Universal Robots PolyScope program: Swan.urp

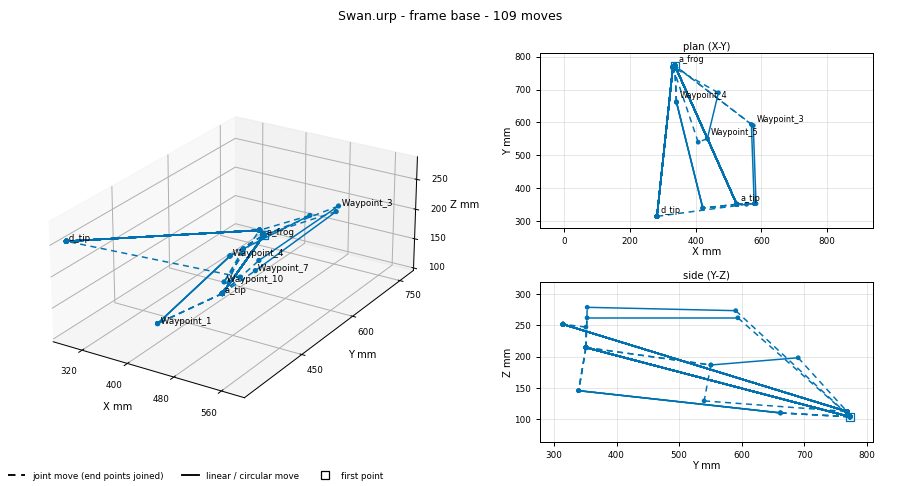
[picture p0: tool path of Swan.urp in frame base, 109 of 109 moves have a stored position in this frame; points joined in program order, loops and branches not executed]
Program Swan (installation=string_planes directory=/programs createdIn=5.17.3 lastSavedIn=5.17.3 robotSerialNumber=20245501435)
Calibrated DH parameters: a=[0.000154, -0.137004, -0.385524, -0.00002, 0.000092, 0]; d=[0.162441, 211.794786, -230.585024, 18.923638, 0.099786, 0.09951]; alpha=[1.569493, -0.001902, 0.003874, 1.570111, -1.570167, 0]; deltaTheta=[0, -1.242934, 1.056292, 0.186646, 0.000002, 0.000001]
InitVariablesNode
Robot Program (runOnlyOnce=true)
  SuppressedNode
    Wait Sleep waitTime=20
  Timer (action=Start) variable(name=beats)
  MoveL speed 150 mm/s, acceleration 600 mm/s^2 (useActiveTCP=true) feature=Base
    Waypoint a_frog: TCP in base x=336.638 y=773.336 z=103.937 mm, rx=-1.3698 ry=-2.3362 rz=1.327 rad; joints [-127.102, -6.181, 18.995, -50.118, -88.699, -156.884] deg; TCP offset x=28.21 y=-96.107 z=-99.69 mm, rx=0 ry=0 rz=0 rad
    Waypoint a_tip: TCP in base x=525.206 y=350.983 z=214.78 mm, rx=-1.3698 ry=-2.3362 rz=1.327 rad; joints [-161.028, -44.56, 81.191, -78.693, -115.03, -178.818] deg
      Until EXPRESSION (allowActions=false) ExpressionBranch=beats≥3
    Timer (action=Reset) variable=beats
  MoveJ speed 60 deg/s, acceleration 80 deg/s^2 (useActiveTCP=true) feature=Base
    Waypoint Waypoint_1: TCP in base x=421.786 y=339.391 z=145.77 mm, rx=-1.4848 ry=-2.1696 rz=1.0787 rad; joints [-159.235, -47.179, 101.918, -97.789, -99.401, -176.138] deg
  Timer (action=Reset) variable=beats
  MoveL speed 150 mm/s, acceleration 500 mm/s^2 (useActiveTCP=true) feature=Base
    Waypoint Waypoint_4: TCP in base x=341.564 y=662.071 z=110.192 mm, rx=-1.458 ry=-2.1893 rz=0.9879 rad; joints [-132.282, -25.96, 62.515, -82.619, -77.894, -159.669] deg
      Until EXPRESSION (allowActions=false) ExpressionBranch=beats≥3
  MoveJ speed 60 deg/s, acceleration 80 deg/s^2 (useActiveTCP=true) feature=Base
    Waypoint a_frog: TCP in base x=336.638 y=773.336 z=103.937 mm, rx=-1.3698 ry=-2.3362 rz=1.327 rad; joints [-127.102, -6.181, 18.995, -50.118, -88.699, -156.884] deg
  Timer (action=Reset) variable=beats
  MoveL speed 100 mm/s, acceleration 300 mm/s^2 (useActiveTCP=true) feature=Base
    Waypoint a_tip: motionParameters(blendRadius=0.03); TCP in base x=525.206 y=350.983 z=214.78 mm, rx=-1.3698 ry=-2.3362 rz=1.327 rad; joints [-161.028, -44.56, 81.191, -78.693, -115.03, -178.818] deg
      Until EXPRESSION (allowActions=false) ExpressionBranch=beats≥2.5
  Timer (action=Reset) variable=beats
  MoveL speed 400 mm/s, acceleration 1200 mm/s^2 (useActiveTCP=true) feature=Base
    Waypoint a_frog: TCP in base x=336.638 y=773.336 z=103.937 mm, rx=-1.3698 ry=-2.3362 rz=1.327 rad; joints [-127.102, -6.181, 18.995, -50.118, -88.699, -156.884] deg
      Until EXPRESSION (allowActions=false) ExpressionBranch=beats≥0.5
  Timer (action=Reset) variable=beats
  MoveL speed 100 mm/s, acceleration 600 mm/s^2 (useActiveTCP=true) feature=Base
    Waypoint a_tip: motionParameters(blendRadius=0.03); TCP in base x=525.206 y=350.983 z=214.78 mm, rx=-1.3698 ry=-2.3362 rz=1.327 rad; joints [-161.028, -44.56, 81.191, -78.693, -115.03, -178.818] deg
      Until EXPRESSION (allowActions=false) ExpressionBranch=beats≥2
  SuppressedNode
    Wait Sleep waitTime=21
  MoveJ speed 60 deg/s, acceleration 80 deg/s^2 (useActiveTCP=true) feature=Base
    Waypoint Waypoint_5: TCP in base x=435.657 y=550.869 z=186.821 mm, rx=-1.3927 ry=-2.3599 rz=1.285 rad; joints [-143.387, -35.735, 67.715, -72.278, -101.384, -166.853] deg
  MoveJ speed 60 deg/s, acceleration 80 deg/s^2 (useActiveTCP=true) feature=Base
    Waypoint Waypoint_10: TCP in base x=407.775 y=540.024 z=129.396 mm, rx=-1.4447 ry=-1.9576 rz=1.0842 rad; joints [-142.798, -34.554, 77.92, -79.333, -77.889, -165.949] deg
  SuppressedNode
    MoveL speed 400 mm/s, acceleration 1200 mm/s^2 (useActiveTCP=true) feature=Base
      Waypoint Waypoint_6: TCP in base x=469.305 y=690.432 z=198.38 mm, rx=-1.3698 ry=-2.3362 rz=1.327 rad; joints [-137.273, -11.027, 15.189, -41.782, -96.797, -163.098] deg
  MoveJ speed 60 deg/s, acceleration 80 deg/s^2 (useActiveTCP=true) feature=Base
    Waypoint d_frog: TCP in base x=330.848 y=768.457 z=112.523 mm, rx=-1.919 ry=-1.7189 rz=1.2902 rad; joints [-128.404, -20.72, 47.39, -64.46, -68.674, -132.513] deg
  Timer (action=Reset) variable=beats
  MoveL speed 200 mm/s, acceleration 600 mm/s^2 (useActiveTCP=true) feature=Base
    Waypoint d_tip: TCP in base x=282.292 y=314.303 z=251.965 mm, rx=-1.8973 ry=-1.7705 rz=1.2029 rad; joints [-160.183, -75.446, 125.19, -87.671, -93.352, -154.437] deg
      Until EXPRESSION (allowActions=false) ExpressionBranch=beats≥2
  Timer (action=Reset) variable=beats
  Timer (action=Start) variable=beats
  MoveL speed 150 mm/s, acceleration 600 mm/s^2 (useActiveTCP=true) feature=Base
    Waypoint d_frog: TCP in base x=330.848 y=768.457 z=112.523 mm, rx=-1.919 ry=-1.7189 rz=1.2902 rad; joints [-128.404, -20.72, 47.39, -64.46, -68.674, -132.513] deg
      Until EXPRESSION (allowActions=false) ExpressionBranch=beats≥0.5
  Timer (action=Reset) variable=beats
  MoveL speed 150 mm/s, acceleration 600 mm/s^2 (useActiveTCP=true) feature=Base
    Waypoint d_tip: TCP in base x=282.292 y=314.303 z=251.965 mm, rx=-1.8973 ry=-1.7705 rz=1.2029 rad; joints [-160.183, -75.446, 125.19, -87.671, -93.352, -154.437] deg
      Until EXPRESSION (allowActions=false) ExpressionBranch=beats≥0.5
  Timer (action=Reset) variable=beats
  MoveL speed 150 mm/s, acceleration 600 mm/s^2 (useActiveTCP=true) feature=Base
    Waypoint d_frog: TCP in base x=330.848 y=768.457 z=112.523 mm, rx=-1.919 ry=-1.7189 rz=1.2902 rad; joints [-128.404, -20.72, 47.39, -64.46, -68.674, -132.513] deg
      Until EXPRESSION (allowActions=false) ExpressionBranch=beats≥0.5
  Timer (action=Reset) variable=beats
  MoveL speed 150 mm/s, acceleration 600 mm/s^2 (useActiveTCP=true) feature=Base
    Waypoint d_tip: TCP in base x=282.292 y=314.303 z=251.965 mm, rx=-1.8973 ry=-1.7705 rz=1.2029 rad; joints [-160.183, -75.446, 125.19, -87.671, -93.352, -154.437] deg
      Until EXPRESSION (allowActions=false) ExpressionBranch=beats≥0.5
  Timer (action=Reset) variable=beats
  MoveL speed 150 mm/s, acceleration 600 mm/s^2 (useActiveTCP=true) feature=Base
    Waypoint d_frog: TCP in base x=330.848 y=768.457 z=112.523 mm, rx=-1.919 ry=-1.7189 rz=1.2902 rad; joints [-128.404, -20.72, 47.39, -64.46, -68.674, -132.513] deg
      Until EXPRESSION (allowActions=false) ExpressionBranch=beats≥0.5
  Timer (action=Reset) variable=beats
  MoveL speed 150 mm/s, acceleration 600 mm/s^2 (useActiveTCP=true) feature=Base
    Waypoint d_tip: TCP in base x=282.292 y=314.303 z=251.965 mm, rx=-1.8973 ry=-1.7705 rz=1.2029 rad; joints [-160.183, -75.446, 125.19, -87.671, -93.352, -154.437] deg
      Until EXPRESSION (allowActions=false) ExpressionBranch=beats≥0.5
  Timer (action=Reset) variable=beats
  MoveL speed 150 mm/s, acceleration 600 mm/s^2 (useActiveTCP=true) feature=Base
    Waypoint d_frog: TCP in base x=330.848 y=768.457 z=112.523 mm, rx=-1.919 ry=-1.7189 rz=1.2902 rad; joints [-128.404, -20.72, 47.39, -64.46, -68.674, -132.513] deg
      Until EXPRESSION (allowActions=false) ExpressionBranch=beats≥0.5
  Timer (action=Reset) variable=beats
  MoveL speed 150 mm/s, acceleration 600 mm/s^2 (useActiveTCP=true) feature=Base
    Waypoint d_tip: TCP in base x=282.292 y=314.303 z=251.965 mm, rx=-1.8973 ry=-1.7705 rz=1.2029 rad; joints [-160.183, -75.446, 125.19, -87.671, -93.352, -154.437] deg
      Until EXPRESSION (allowActions=false) ExpressionBranch=beats≥0.5
  Timer (action=Reset) variable=beats
  MoveL speed 150 mm/s, acceleration 600 mm/s^2 (useActiveTCP=true) feature=Base
    Waypoint d_frog: TCP in base x=330.848 y=768.457 z=112.523 mm, rx=-1.919 ry=-1.7189 rz=1.2902 rad; joints [-128.404, -20.72, 47.39, -64.46, -68.674, -132.513] deg
      Until EXPRESSION (allowActions=false) ExpressionBranch=beats≥3.5
  MoveJ speed 60 deg/s, acceleration 80 deg/s^2 (useActiveTCP=true) feature=Base
    Waypoint a_frog: TCP in base x=336.638 y=773.336 z=103.937 mm, rx=-1.3698 ry=-2.3362 rz=1.327 rad; joints [-127.102, -6.181, 18.995, -50.118, -88.699, -156.884] deg
  Wait Sleep waitTime=1
  Timer (action=Reset) variable=beats
  MoveL speed 150 mm/s, acceleration 600 mm/s^2 (useActiveTCP=true) feature=Base
    Waypoint a_frog: TCP in base x=336.638 y=773.336 z=103.937 mm, rx=-1.3698 ry=-2.3362 rz=1.327 rad; joints [-127.102, -6.181, 18.995, -50.118, -88.699, -156.884] deg
    Waypoint a_tip: TCP in base x=525.206 y=350.983 z=214.78 mm, rx=-1.3698 ry=-2.3362 rz=1.327 rad; joints [-161.028, -44.56, 81.191, -78.693, -115.03, -178.818] deg
      Until EXPRESSION (allowActions=false) ExpressionBranch=beats≥3
    Timer (action=Reset) variable=beats
  MoveJ speed 60 deg/s, acceleration 80 deg/s^2 (useActiveTCP=true) feature=Base
    Waypoint Waypoint_1: TCP in base x=421.786 y=339.391 z=145.77 mm, rx=-1.4848 ry=-2.1696 rz=1.0787 rad; joints [-159.235, -47.179, 101.918, -97.789, -99.401, -176.138] deg
  Timer (action=Reset) variable=beats
  MoveL speed 150 mm/s, acceleration 500 mm/s^2 (useActiveTCP=true) feature=Base
    Waypoint Waypoint_4: TCP in base x=341.564 y=662.071 z=110.192 mm, rx=-1.458 ry=-2.1893 rz=0.9879 rad; joints [-132.282, -25.96, 62.515, -82.619, -77.894, -159.669] deg
      Until EXPRESSION (allowActions=false) ExpressionBranch=beats≥3
  MoveJ speed 60 deg/s, acceleration 80 deg/s^2 (useActiveTCP=true) feature=Base
    Waypoint a_frog: TCP in base x=336.638 y=773.336 z=103.937 mm, rx=-1.3698 ry=-2.3362 rz=1.327 rad; joints [-127.102, -6.181, 18.995, -50.118, -88.699, -156.884] deg
  MoveL speed 100 mm/s, acceleration 300 mm/s^2 (useActiveTCP=true) feature=Base
    Waypoint a_tip: motionParameters(blendRadius=0.03); TCP in base x=525.206 y=350.983 z=214.78 mm, rx=-1.3698 ry=-2.3362 rz=1.327 rad; joints [-161.028, -44.56, 81.191, -78.693, -115.03, -178.818] deg
      Until EXPRESSION (allowActions=false) ExpressionBranch=beats≥2.5
  Timer (action=Reset) variable=beats
  MoveL speed 250 mm/s, acceleration 1200 mm/s^2 (useActiveTCP=true) feature=Base
    Waypoint a_frog: TCP in base x=336.638 y=773.336 z=103.937 mm, rx=-1.3698 ry=-2.3362 rz=1.327 rad; joints [-127.102, -6.181, 18.995, -50.118, -88.699, -156.884] deg
      Until EXPRESSION (allowActions=false) ExpressionBranch=beats≥0.5
  Timer (action=Reset) variable=beats
  MoveL speed 100 mm/s, acceleration 600 mm/s^2 (useActiveTCP=true) feature=Base
    Waypoint a_tip: motionParameters(blendRadius=0.03); TCP in base x=525.206 y=350.983 z=214.78 mm, rx=-1.3698 ry=-2.3362 rz=1.327 rad; joints [-161.028, -44.56, 81.191, -78.693, -115.03, -178.818] deg
      Until EXPRESSION (allowActions=false) ExpressionBranch=beats≥3
  MoveJ speed 60 deg/s, acceleration 80 deg/s^2 (useActiveTCP=true) feature=Base
    Waypoint Waypoint_9: TCP in base x=554.848 y=350.983 z=247.422 mm, rx=-1.3698 ry=-2.3362 rz=1.327 rad; joints [-161.804, -44.051, 74.534, -72.804, -115.615, -179.417] deg
  MoveJ speed 60 deg/s, acceleration 80 deg/s^2 (useActiveTCP=true) feature=Base
    Waypoint d_tip: TCP in base x=282.292 y=314.303 z=251.965 mm, rx=-1.8973 ry=-1.7705 rz=1.2029 rad; joints [-160.183, -75.446, 125.19, -87.671, -93.352, -154.437] deg
  Timer (action=Reset) variable=beats
  Timer (action=Start) variable=beats
  MoveL speed 150 mm/s, acceleration 60 mm/s^2 (useActiveTCP=true) feature=Base
    Waypoint d_frog: TCP in base x=330.848 y=768.457 z=112.523 mm, rx=-1.919 ry=-1.7189 rz=1.2902 rad; joints [-128.404, -20.72, 47.39, -64.46, -68.674, -132.513] deg
      Until EXPRESSION (allowActions=false) ExpressionBranch=beats≥1.5
  Timer (action=Reset) variable=beats
  Timer (action=Start) variable=beats
  MoveL speed 150 mm/s, acceleration 600 mm/s^2 (useActiveTCP=true) feature=Base
    Waypoint d_tip: TCP in base x=282.292 y=314.303 z=251.965 mm, rx=-1.8973 ry=-1.7705 rz=1.2029 rad; joints [-160.183, -75.446, 125.19, -87.671, -93.352, -154.437] deg
      Until EXPRESSION (allowActions=false) ExpressionBranch=beats≥0.5
  Timer (action=Reset) variable=beats
  MoveL speed 150 mm/s, acceleration 600 mm/s^2 (useActiveTCP=true) feature=Base
    Waypoint d_frog: TCP in base x=330.848 y=768.457 z=112.523 mm, rx=-1.919 ry=-1.7189 rz=1.2902 rad; joints [-128.404, -20.72, 47.39, -64.46, -68.674, -132.513] deg
      Until EXPRESSION (allowActions=false) ExpressionBranch=beats≥0.5
  Timer (action=Reset) variable=beats
  MoveL speed 150 mm/s, acceleration 600 mm/s^2 (useActiveTCP=true) feature=Base
    Waypoint d_tip: TCP in base x=282.292 y=314.303 z=251.965 mm, rx=-1.8973 ry=-1.7705 rz=1.2029 rad; joints [-160.183, -75.446, 125.19, -87.671, -93.352, -154.437] deg
      Until EXPRESSION (allowActions=false) ExpressionBranch=beats≥0.5
  Timer (action=Reset) variable=beats
  MoveL speed 150 mm/s, acceleration 600 mm/s^2 (useActiveTCP=true) feature=Base
    Waypoint d_frog: TCP in base x=330.848 y=768.457 z=112.523 mm, rx=-1.919 ry=-1.7189 rz=1.2902 rad; joints [-128.404, -20.72, 47.39, -64.46, -68.674, -132.513] deg
      Until EXPRESSION (allowActions=false) ExpressionBranch=beats≥0.5
  Timer (action=Reset) variable=beats
  MoveL speed 150 mm/s, acceleration 600 mm/s^2 (useActiveTCP=true) feature=Base
    Waypoint d_tip: TCP in base x=282.292 y=314.303 z=251.965 mm, rx=-1.8973 ry=-1.7705 rz=1.2029 rad; joints [-160.183, -75.446, 125.19, -87.671, -93.352, -154.437] deg
      Until EXPRESSION (allowActions=false) ExpressionBranch=beats≥0.5
  Timer (action=Reset) variable=beats
  MoveL speed 150 mm/s, acceleration 600 mm/s^2 (useActiveTCP=true) feature=Base
    Waypoint d_frog: TCP in base x=330.848 y=768.457 z=112.523 mm, rx=-1.919 ry=-1.7189 rz=1.2902 rad; joints [-128.404, -20.72, 47.39, -64.46, -68.674, -132.513] deg
      Until EXPRESSION (allowActions=false) ExpressionBranch=beats≥0.5
  Timer (action=Reset) variable=beats
  MoveL speed 150 mm/s, acceleration 600 mm/s^2 (useActiveTCP=true) feature=Base
    Waypoint d_tip: TCP in base x=282.292 y=314.303 z=251.965 mm, rx=-1.8973 ry=-1.7705 rz=1.2029 rad; joints [-160.183, -75.446, 125.19, -87.671, -93.352, -154.437] deg
      Until EXPRESSION (allowActions=false) ExpressionBranch=beats≥0.5
  Timer (action=Reset) variable=beats
  MoveL speed 150 mm/s, acceleration 600 mm/s^2 (useActiveTCP=true) feature=Base
    Waypoint d_frog: TCP in base x=330.848 y=768.457 z=112.523 mm, rx=-1.919 ry=-1.7189 rz=1.2902 rad; joints [-128.404, -20.72, 47.39, -64.46, -68.674, -132.513] deg
      Until EXPRESSION (allowActions=false) ExpressionBranch=beats≥0.5
  Timer (action=Reset) variable=beats
  MoveL speed 100 mm/s, acceleration 500 mm/s^2 (useActiveTCP=true) feature=Base
    Waypoint d_frog: TCP in base x=330.848 y=768.457 z=112.523 mm, rx=-1.919 ry=-1.7189 rz=1.2902 rad; joints [-128.404, -20.72, 47.39, -64.46, -68.674, -132.513] deg
      Until EXPRESSION (allowActions=false) ExpressionBranch=beats≥3.5
  MoveJ speed 60 deg/s, acceleration 80 deg/s^2 (useActiveTCP=true) feature=Base
    Waypoint a_frog: TCP in base x=336.638 y=773.336 z=103.937 mm, rx=-1.3698 ry=-2.3362 rz=1.327 rad; joints [-127.102, -6.181, 18.995, -50.118, -88.699, -156.884] deg
  Wait Sleep waitTime=1
  Timer (action=Reset) variable=beats
  MoveL speed 150 mm/s, acceleration 600 mm/s^2 (useActiveTCP=true) feature=Base
    Waypoint a_frog: TCP in base x=336.638 y=773.336 z=103.937 mm, rx=-1.3698 ry=-2.3362 rz=1.327 rad; joints [-127.102, -6.181, 18.995, -50.118, -88.699, -156.884] deg
    Waypoint a_tip: TCP in base x=525.206 y=350.983 z=214.78 mm, rx=-1.3698 ry=-2.3362 rz=1.327 rad; joints [-161.028, -44.56, 81.191, -78.693, -115.03, -178.818] deg
      Until EXPRESSION (allowActions=false) ExpressionBranch=beats≥3
    Timer (action=Reset) variable=beats
  MoveL speed 100 mm/s, acceleration 600 mm/s^2 (useActiveTCP=true) feature=Base
    Waypoint a_frog: TCP in base x=336.638 y=773.336 z=103.937 mm, rx=-1.3698 ry=-2.3362 rz=1.327 rad; joints [-127.102, -6.181, 18.995, -50.118, -88.699, -156.884] deg
      Until EXPRESSION (allowActions=false) ExpressionBranch=beats≥3
  Timer (action=Reset) variable=beats
  MoveL speed 100 mm/s, acceleration 600 mm/s^2 (useActiveTCP=true) feature=Base
    Waypoint a_tip: TCP in base x=525.206 y=350.983 z=214.78 mm, rx=-1.3698 ry=-2.3362 rz=1.327 rad; joints [-161.028, -44.56, 81.191, -78.693, -115.03, -178.818] deg
      Until EXPRESSION (allowActions=false) ExpressionBranch=beats≥2.5
  Timer (action=Reset) variable=beats
  MoveL speed 300 mm/s, acceleration 1200 mm/s^2 (useActiveTCP=true) feature=Base
    Waypoint a_frog: TCP in base x=336.638 y=773.336 z=103.937 mm, rx=-1.3698 ry=-2.3362 rz=1.327 rad; joints [-127.102, -6.181, 18.995, -50.118, -88.699, -156.884] deg
      Until EXPRESSION (allowActions=false) ExpressionBranch=beats≥0.5
  MoveL speed 150 mm/s, acceleration 600 mm/s^2 (useActiveTCP=true) feature=Base
    Waypoint a_tip: TCP in base x=525.206 y=350.983 z=214.78 mm, rx=-1.3698 ry=-2.3362 rz=1.327 rad; joints [-161.028, -44.56, 81.191, -78.693, -115.03, -178.818] deg
      Until EXPRESSION (allowActions=false) ExpressionBranch=beats≥2
  MoveJ speed 60 deg/s, acceleration 80 deg/s^2 (useActiveTCP=true) feature=Base
    Waypoint Waypoint_2: TCP in base x=583.831 y=353.076 z=279.049 mm, rx=-1.3698 ry=-2.3362 rz=1.327 rad; joints [-162.353, -42.73, 66.875, -66.655, -116.033, -179.849] deg
  MoveL speed 400 mm/s, acceleration 1200 mm/s^2 (useActiveTCP=true) feature=Base
    Waypoint Waypoint_3: TCP in base x=575.353 y=590.579 z=273.677 mm, rx=-1.3698 ry=-2.3362 rz=1.327 rad; joints [-146.762, -11.123, 4.55, -32.162, -104.295, -169.078] deg
  MoveJ speed 60 deg/s, acceleration 80 deg/s^2 (useActiveTCP=true) feature=Base
    Waypoint a_frog: TCP in base x=336.638 y=773.336 z=103.937 mm, rx=-1.3698 ry=-2.3362 rz=1.327 rad; joints [-127.102, -6.181, 18.995, -50.118, -88.699, -156.884] deg
  MoveL speed 200 mm/s, acceleration 600 mm/s^2 (useActiveTCP=true) feature=Base
    Waypoint a_tip: TCP in base x=525.206 y=350.983 z=214.78 mm, rx=-1.3698 ry=-2.3362 rz=1.327 rad; joints [-161.028, -44.56, 81.191, -78.693, -115.03, -178.818] deg
      Until EXPRESSION (allowActions=false) ExpressionBranch=beats≥1
  Timer (action=Reset) variable=beats
  MoveL speed 200 mm/s, acceleration 600 mm/s^2 (useActiveTCP=true) feature=Base
    Waypoint a_frog: TCP in base x=336.638 y=773.336 z=103.937 mm, rx=-1.3698 ry=-2.3362 rz=1.327 rad; joints [-127.102, -6.181, 18.995, -50.118, -88.699, -156.884] deg
      Until EXPRESSION (allowActions=false) ExpressionBranch=beats≥1
  Timer (action=Reset) variable=beats
  MoveL speed 200 mm/s, acceleration 600 mm/s^2 (useActiveTCP=true) feature=Base
    Waypoint a_tip: TCP in base x=525.206 y=350.983 z=214.78 mm, rx=-1.3698 ry=-2.3362 rz=1.327 rad; joints [-161.028, -44.56, 81.191, -78.693, -115.03, -178.818] deg
      Until EXPRESSION (allowActions=false) ExpressionBranch=beats≥1
  Timer (action=Reset) variable=beats
  MoveL speed 200 mm/s, acceleration 600 mm/s^2 (useActiveTCP=true) feature=Base
    Waypoint a_frog: TCP in base x=336.638 y=773.336 z=103.937 mm, rx=-1.3698 ry=-2.3362 rz=1.327 rad; joints [-127.102, -6.181, 18.995, -50.118, -88.699, -156.884] deg
      Until EXPRESSION (allowActions=false) ExpressionBranch=beats≥1
  Timer (action=Reset) variable=beats
  MoveL speed 200 mm/s, acceleration 600 mm/s^2 (useActiveTCP=true) feature=Base
    Waypoint a_tip: TCP in base x=525.206 y=350.983 z=214.78 mm, rx=-1.3698 ry=-2.3362 rz=1.327 rad; joints [-161.028, -44.56, 81.191, -78.693, -115.03, -178.818] deg
      Until EXPRESSION (allowActions=false) ExpressionBranch=beats≥1
  Timer (action=Reset) variable=beats
  MoveL speed 250 mm/s, acceleration 600 mm/s^2 (useActiveTCP=true) feature=Base
    Waypoint a_frog: TCP in base x=336.638 y=773.336 z=103.937 mm, rx=-1.3698 ry=-2.3362 rz=1.327 rad; joints [-127.102, -6.181, 18.995, -50.118, -88.699, -156.884] deg
      Until EXPRESSION (allowActions=false) ExpressionBranch=beats≥1
  Timer (action=Reset) variable=beats
  MoveL speed 100 mm/s, acceleration 600 mm/s^2 (useActiveTCP=true) feature=Base
    Waypoint a_tip: TCP in base x=525.206 y=350.983 z=214.78 mm, rx=-1.3698 ry=-2.3362 rz=1.327 rad; joints [-161.028, -44.56, 81.191, -78.693, -115.03, -178.818] deg
      Until EXPRESSION (allowActions=false) ExpressionBranch=beats≥2.5
  Timer (action=Reset) variable=beats
  MoveL speed 250 mm/s, acceleration 1200 mm/s^2 (useActiveTCP=true) feature=Base
    Waypoint a_frog: TCP in base x=336.638 y=773.336 z=103.937 mm, rx=-1.3698 ry=-2.3362 rz=1.327 rad; joints [-127.102, -6.181, 18.995, -50.118, -88.699, -156.884] deg
      Until EXPRESSION (allowActions=false) ExpressionBranch=beats≥0.5
  Timer (action=Reset) variable=beats
  MoveL speed 150 mm/s, acceleration 600 mm/s^2 (useActiveTCP=true) feature=Base
    Waypoint a_tip: TCP in base x=525.206 y=350.983 z=214.78 mm, rx=-1.3698 ry=-2.3362 rz=1.327 rad; joints [-161.028, -44.56, 81.191, -78.693, -115.03, -178.818] deg
      Until EXPRESSION (allowActions=false) ExpressionBranch=beats≥2
  Timer (action=Reset) variable=beats
  MoveJ speed 60 deg/s, acceleration 80 deg/s^2 (useActiveTCP=true) feature=Base
    Waypoint Waypoint_7: TCP in base x=578.283 y=352.878 z=262.264 mm, rx=-1.3698 ry=-2.3362 rz=1.327 rad; joints [-162.237, -42.346, 68.857, -68.978, -115.943, -179.753] deg
  MoveL speed 400 mm/s, acceleration 1200 mm/s^2 (useActiveTCP=true) feature=Base
    Waypoint Waypoint_8: TCP in base x=569.678 y=593.931 z=262.264 mm, rx=-1.3698 ry=-2.3362 rz=1.327 rad; joints [-146.374, -13.725, 11.576, -36.522, -103.973, -168.824] deg
  MoveJ speed 60 deg/s, acceleration 80 deg/s^2 (useActiveTCP=true) feature=Base
    Waypoint a_frog: TCP in base x=336.638 y=773.336 z=103.937 mm, rx=-1.3698 ry=-2.3362 rz=1.327 rad; joints [-127.102, -6.181, 18.995, -50.118, -88.699, -156.884] deg
  Timer (action=Reset) variable=beats
  MoveL speed 200 mm/s, acceleration 600 mm/s^2 (useActiveTCP=true) feature=Base
    Waypoint a_tip: TCP in base x=525.206 y=350.983 z=214.78 mm, rx=-1.3698 ry=-2.3362 rz=1.327 rad; joints [-161.028, -44.56, 81.191, -78.693, -115.03, -178.818] deg
      Until EXPRESSION (allowActions=false) ExpressionBranch=beats≥1
  Timer (action=Reset) variable=beats
  MoveL speed 200 mm/s, acceleration 600 mm/s^2 (useActiveTCP=true) feature=Base
    Waypoint a_frog: TCP in base x=336.638 y=773.336 z=103.937 mm, rx=-1.3698 ry=-2.3362 rz=1.327 rad; joints [-127.102, -6.181, 18.995, -50.118, -88.699, -156.884] deg
      Until EXPRESSION (allowActions=false) ExpressionBranch=beats≥1
  Timer (action=Reset) variable=beats
  MoveL speed 200 mm/s, acceleration 600 mm/s^2 (useActiveTCP=true) feature=Base
    Waypoint a_tip: TCP in base x=525.206 y=350.983 z=214.78 mm, rx=-1.3698 ry=-2.3362 rz=1.327 rad; joints [-161.028, -44.56, 81.191, -78.693, -115.03, -178.818] deg
      Until EXPRESSION (allowActions=false) ExpressionBranch=beats≥1
  Timer (action=Reset) variable=beats
  MoveL speed 100 mm/s, acceleration 600 mm/s^2 (useActiveTCP=true) feature=Base
    Waypoint a_frog: TCP in base x=336.638 y=773.336 z=103.937 mm, rx=-1.3698 ry=-2.3362 rz=1.327 rad; joints [-127.102, -6.181, 18.995, -50.118, -88.699, -156.884] deg
      Until EXPRESSION (allowActions=false) ExpressionBranch=beats≥2
  Timer (action=Reset) variable=beats
  MoveL speed 250 mm/s, acceleration 1200 mm/s^2 (useActiveTCP=true) feature=Base
    Waypoint a_tip: TCP in base x=525.206 y=350.983 z=214.78 mm, rx=-1.3698 ry=-2.3362 rz=1.327 rad; joints [-161.028, -44.56, 81.191, -78.693, -115.03, -178.818] deg
      Until EXPRESSION (allowActions=false) ExpressionBranch=beats≥0.5
  Timer (action=Reset) variable=beats
  MoveL speed 250 mm/s, acceleration 1200 mm/s^2 (useActiveTCP=true) feature=Base
    Waypoint a_frog: TCP in base x=336.638 y=773.336 z=103.937 mm, rx=-1.3698 ry=-2.3362 rz=1.327 rad; joints [-127.102, -6.181, 18.995, -50.118, -88.699, -156.884] deg
      Until EXPRESSION (allowActions=false) ExpressionBranch=beats≥0.5
  Timer (action=Reset) variable=beats
  MoveL speed 150 mm/s, acceleration 600 mm/s^2 (useActiveTCP=true) feature=Base
    Waypoint a_tip: TCP in base x=525.206 y=350.983 z=214.78 mm, rx=-1.3698 ry=-2.3362 rz=1.327 rad; joints [-161.028, -44.56, 81.191, -78.693, -115.03, -178.818] deg
      Until EXPRESSION (allowActions=false) ExpressionBranch=beats≥3
  Timer (action=Reset) variable=beats
  MoveL speed 150 mm/s, acceleration 600 mm/s^2 (useActiveTCP=true) feature=Base
    Waypoint a_frog: TCP in base x=336.638 y=773.336 z=103.937 mm, rx=-1.3698 ry=-2.3362 rz=1.327 rad; joints [-127.102, -6.181, 18.995, -50.118, -88.699, -156.884] deg
      Until EXPRESSION (allowActions=false) ExpressionBranch=beats≥3
  Timer (action=Reset) variable=beats
  MoveL speed 150 mm/s, acceleration 600 mm/s^2 (useActiveTCP=true) feature=Base
    Waypoint a_tip: TCP in base x=525.206 y=350.983 z=214.78 mm, rx=-1.3698 ry=-2.3362 rz=1.327 rad; joints [-161.028, -44.56, 81.191, -78.693, -115.03, -178.818] deg
      Until EXPRESSION (allowActions=false) ExpressionBranch=beats≥3
  Timer (action=Reset) variable=beats
  MoveL speed 150 mm/s, acceleration 600 mm/s^2 (useActiveTCP=true) feature=Base
    Waypoint a_frog: TCP in base x=336.638 y=773.336 z=103.937 mm, rx=-1.3698 ry=-2.3362 rz=1.327 rad; joints [-127.102, -6.181, 18.995, -50.118, -88.699, -156.884] deg
      Until EXPRESSION (allowActions=false) ExpressionBranch=beats≥2
  Timer (action=Reset) variable=beats
  MoveL speed 250 mm/s, acceleration 1200 mm/s^2 (useActiveTCP=true) feature=Base
    Waypoint a_tip: TCP in base x=525.206 y=350.983 z=214.78 mm, rx=-1.3698 ry=-2.3362 rz=1.327 rad; joints [-161.028, -44.56, 81.191, -78.693, -115.03, -178.818] deg
      Until EXPRESSION (allowActions=false) ExpressionBranch=beats≥0.5
  Timer (action=Reset) variable=beats
  MoveL speed 250 mm/s, acceleration 1200 mm/s^2 (useActiveTCP=true) feature=Base
    Waypoint a_frog: TCP in base x=336.638 y=773.336 z=103.937 mm, rx=-1.3698 ry=-2.3362 rz=1.327 rad; joints [-127.102, -6.181, 18.995, -50.118, -88.699, -156.884] deg
      Until EXPRESSION (allowActions=false) ExpressionBranch=beats≥0.5
  Timer (action=Reset) variable=beats
  MoveL speed 150 mm/s, acceleration 600 mm/s^2 (useActiveTCP=true) feature=Base
    Waypoint a_tip: TCP in base x=525.206 y=350.983 z=214.78 mm, rx=-1.3698 ry=-2.3362 rz=1.327 rad; joints [-161.028, -44.56, 81.191, -78.693, -115.03, -178.818] deg
      Until EXPRESSION (allowActions=false) ExpressionBranch=beats≥3
  Timer (action=Reset) variable=beats
  MoveL speed 150 mm/s, acceleration 600 mm/s^2 (useActiveTCP=true) feature=Base
    Waypoint a_frog: TCP in base x=336.638 y=773.336 z=103.937 mm, rx=-1.3698 ry=-2.3362 rz=1.327 rad; joints [-127.102, -6.181, 18.995, -50.118, -88.699, -156.884] deg
      Until EXPRESSION (allowActions=false) ExpressionBranch=beats≥3
  Timer (action=Reset) variable=beats
  MoveL speed 150 mm/s, acceleration 600 mm/s^2 (useActiveTCP=true) feature=Base
    Waypoint a_tip: TCP in base x=525.206 y=350.983 z=214.78 mm, rx=-1.3698 ry=-2.3362 rz=1.327 rad; joints [-161.028, -44.56, 81.191, -78.693, -115.03, -178.818] deg
      Until EXPRESSION (allowActions=false) ExpressionBranch=beats≥3
    Timer (action=Reset) variable=beats
  MoveJ speed 60 deg/s, acceleration 80 deg/s^2 (useActiveTCP=true) feature=Base
    Waypoint Waypoint_1: motionParameters(blendRadius=0.03); TCP in base x=421.786 y=339.391 z=145.77 mm, rx=-1.4848 ry=-2.1696 rz=1.0787 rad; joints [-159.235, -47.179, 101.918, -97.789, -99.401, -176.138] deg
  Timer (action=Reset) variable=beats
  MoveL speed 150 mm/s, acceleration 500 mm/s^2 (useActiveTCP=true) feature=Base
    Waypoint Waypoint_4: TCP in base x=341.564 y=662.071 z=110.192 mm, rx=-1.458 ry=-2.1893 rz=0.9879 rad; joints [-132.282, -25.96, 62.515, -82.619, -77.894, -159.669] deg
      Until EXPRESSION (allowActions=false) ExpressionBranch=beats≥3
  MoveJ speed 60 deg/s, acceleration 80 deg/s^2 (useActiveTCP=true) feature=Base
    Waypoint a_frog: TCP in base x=336.638 y=773.336 z=103.937 mm, rx=-1.3698 ry=-2.3362 rz=1.327 rad; joints [-127.102, -6.181, 18.995, -50.118, -88.699, -156.884] deg
  Timer (action=Reset) variable=beats
  MoveL speed 150 mm/s, acceleration 300 mm/s^2 (useActiveTCP=true) feature=Base
    Waypoint a_tip: motionParameters(blendRadius=0.03); TCP in base x=525.206 y=350.983 z=214.78 mm, rx=-1.3698 ry=-2.3362 rz=1.327 rad; joints [-161.028, -44.56, 81.191, -78.693, -115.03, -178.818] deg
      Until EXPRESSION (allowActions=false) ExpressionBranch=beats≥2.5
  Timer (action=Reset) variable=beats
  MoveL speed 300 mm/s, acceleration 1200 mm/s^2 (useActiveTCP=true) feature=Base
    Waypoint a_frog: TCP in base x=336.638 y=773.336 z=103.937 mm, rx=-1.3698 ry=-2.3362 rz=1.327 rad; joints [-127.102, -6.181, 18.995, -50.118, -88.699, -156.884] deg
      Until EXPRESSION (allowActions=false) ExpressionBranch=beats≥0.5
  Timer (action=Reset) variable=beats
  MoveL speed 100 mm/s, acceleration 600 mm/s^2 (useActiveTCP=true) feature=Base
    Waypoint a_tip: motionParameters(blendRadius=0.03); TCP in base x=525.206 y=350.983 z=214.78 mm, rx=-1.3698 ry=-2.3362 rz=1.327 rad; joints [-161.028, -44.56, 81.191, -78.693, -115.03, -178.818] deg
      Until EXPRESSION (allowActions=false) ExpressionBranch=beats≥2
  MoveJ speed 60 deg/s, acceleration 80 deg/s^2 (useActiveTCP=true) feature=Base
    Waypoint Waypoint_5: TCP in base x=435.657 y=550.869 z=186.821 mm, rx=-1.3927 ry=-2.3599 rz=1.285 rad; joints [-143.387, -35.735, 67.715, -72.278, -101.384, -166.853] deg
  MoveL speed 400 mm/s, acceleration 1200 mm/s^2 (useActiveTCP=true) feature=Base
    Waypoint Waypoint_6: TCP in base x=469.305 y=690.432 z=198.38 mm, rx=-1.3698 ry=-2.3362 rz=1.327 rad; joints [-137.273, -11.027, 15.189, -41.782, -96.797, -163.098] deg
  MoveJ speed 60 deg/s, acceleration 80 deg/s^2 (useActiveTCP=true) feature=Base
    Waypoint d_frog: TCP in base x=330.848 y=768.457 z=112.523 mm, rx=-1.919 ry=-1.7189 rz=1.2902 rad; joints [-128.404, -20.72, 47.39, -64.46, -68.674, -132.513] deg
  Timer (action=Reset) variable=beats
  MoveL speed 150 mm/s, acceleration 600 mm/s^2 (useActiveTCP=true) feature=Base
    Waypoint d_tip: TCP in base x=282.292 y=314.303 z=251.965 mm, rx=-1.8973 ry=-1.7705 rz=1.2029 rad; joints [-160.183, -75.446, 125.19, -87.671, -93.352, -154.437] deg
      Until EXPRESSION (allowActions=false) ExpressionBranch=beats≥2
  Timer (action=Reset) variable=beats
  Timer (action=Start) variable=beats
  MoveL speed 150 mm/s, acceleration 600 mm/s^2 (useActiveTCP=true) feature=Base
    Waypoint d_frog: TCP in base x=330.848 y=768.457 z=112.523 mm, rx=-1.919 ry=-1.7189 rz=1.2902 rad; joints [-128.404, -20.72, 47.39, -64.46, -68.674, -132.513] deg
      Until EXPRESSION (allowActions=false) ExpressionBranch=beats≥0.5
  Timer (action=Reset) variable=beats
  MoveL speed 150 mm/s, acceleration 600 mm/s^2 (useActiveTCP=true) feature=Base
    Waypoint d_tip: TCP in base x=282.292 y=314.303 z=251.965 mm, rx=-1.8973 ry=-1.7705 rz=1.2029 rad; joints [-160.183, -75.446, 125.19, -87.671, -93.352, -154.437] deg
      Until EXPRESSION (allowActions=false) ExpressionBranch=beats≥0.5
  Timer (action=Reset) variable=beats
  MoveL speed 150 mm/s, acceleration 600 mm/s^2 (useActiveTCP=true) feature=Base
    Waypoint d_frog: TCP in base x=330.848 y=768.457 z=112.523 mm, rx=-1.919 ry=-1.7189 rz=1.2902 rad; joints [-128.404, -20.72, 47.39, -64.46, -68.674, -132.513] deg
      Until EXPRESSION (allowActions=false) ExpressionBranch=beats≥0.5
  Timer (action=Reset) variable=beats
  MoveL speed 150 mm/s, acceleration 600 mm/s^2 (useActiveTCP=true) feature=Base
    Waypoint d_tip: TCP in base x=282.292 y=314.303 z=251.965 mm, rx=-1.8973 ry=-1.7705 rz=1.2029 rad; joints [-160.183, -75.446, 125.19, -87.671, -93.352, -154.437] deg
      Until EXPRESSION (allowActions=false) ExpressionBranch=beats≥0.5
  Timer (action=Reset) variable=beats
  MoveL speed 150 mm/s, acceleration 600 mm/s^2 (useActiveTCP=true) feature=Base
    Waypoint d_frog: TCP in base x=330.848 y=768.457 z=112.523 mm, rx=-1.919 ry=-1.7189 rz=1.2902 rad; joints [-128.404, -20.72, 47.39, -64.46, -68.674, -132.513] deg
      Until EXPRESSION (allowActions=false) ExpressionBranch=beats≥0.5
  Timer (action=Reset) variable=beats
  MoveL speed 150 mm/s, acceleration 600 mm/s^2 (useActiveTCP=true) feature=Base
    Waypoint d_tip: TCP in base x=282.292 y=314.303 z=251.965 mm, rx=-1.8973 ry=-1.7705 rz=1.2029 rad; joints [-160.183, -75.446, 125.19, -87.671, -93.352, -154.437] deg
      Until EXPRESSION (allowActions=false) ExpressionBranch=beats≥0.5
  Timer (action=Reset) variable=beats
  MoveL speed 150 mm/s, acceleration 600 mm/s^2 (useActiveTCP=true) feature=Base
    Waypoint d_frog: TCP in base x=330.848 y=768.457 z=112.523 mm, rx=-1.919 ry=-1.7189 rz=1.2902 rad; joints [-128.404, -20.72, 47.39, -64.46, -68.674, -132.513] deg
      Until EXPRESSION (allowActions=false) ExpressionBranch=beats≥0.5
  Timer (action=Reset) variable=beats
  MoveL speed 150 mm/s, acceleration 600 mm/s^2 (useActiveTCP=true) feature=Base
    Waypoint d_tip: TCP in base x=282.292 y=314.303 z=251.965 mm, rx=-1.8973 ry=-1.7705 rz=1.2029 rad; joints [-160.183, -75.446, 125.19, -87.671, -93.352, -154.437] deg
      Until EXPRESSION (allowActions=false) ExpressionBranch=beats≥0.5
  Timer (action=Reset) variable=beats
  MoveL speed 90 mm/s, acceleration 500 mm/s^2 (useActiveTCP=true) feature=Base
    Waypoint d_frog: TCP in base x=330.848 y=768.457 z=112.523 mm, rx=-1.919 ry=-1.7189 rz=1.2902 rad; joints [-128.404, -20.72, 47.39, -64.46, -68.674, -132.513] deg
      Until EXPRESSION (allowActions=false) ExpressionBranch=beats≥4
  MoveJ speed 60 deg/s, acceleration 80 deg/s^2 (useActiveTCP=true) feature=Base
    Waypoint a_frog: TCP in base x=336.638 y=773.336 z=103.937 mm, rx=-1.3698 ry=-2.3362 rz=1.327 rad; joints [-127.102, -6.181, 18.995, -50.118, -88.699, -156.884] deg
  Timer (action=Reset) variable=beats
  MoveL speed 150 mm/s, acceleration 600 mm/s^2 (useActiveTCP=true) feature=Base
    Waypoint a_frog: TCP in base x=336.638 y=773.336 z=103.937 mm, rx=-1.3698 ry=-2.3362 rz=1.327 rad; joints [-127.102, -6.181, 18.995, -50.118, -88.699, -156.884] deg
    Waypoint a_tip: TCP in base x=525.206 y=350.983 z=214.78 mm, rx=-1.3698 ry=-2.3362 rz=1.327 rad; joints [-161.028, -44.56, 81.191, -78.693, -115.03, -178.818] deg
      Until EXPRESSION (allowActions=false) ExpressionBranch=beats≥3
    Timer (action=Reset) variable=beats
  MoveL speed 100 mm/s, acceleration 600 mm/s^2 (useActiveTCP=true) feature=Base
    Waypoint a_frog: TCP in base x=336.638 y=773.336 z=103.937 mm, rx=-1.3698 ry=-2.3362 rz=1.327 rad; joints [-127.102, -6.181, 18.995, -50.118, -88.699, -156.884] deg
      Until EXPRESSION (allowActions=false) ExpressionBranch=beats≥3
  Timer (action=Reset) variable=beats
  MoveL speed 100 mm/s, acceleration 600 mm/s^2 (useActiveTCP=true) feature=Base
    Waypoint a_tip: TCP in base x=525.206 y=350.983 z=214.78 mm, rx=-1.3698 ry=-2.3362 rz=1.327 rad; joints [-161.028, -44.56, 81.191, -78.693, -115.03, -178.818] deg
      Until EXPRESSION (allowActions=false) ExpressionBranch=beats≥3
    Timer (action=Reset) variable=beats
  MoveL speed 100 mm/s, acceleration 600 mm/s^2 (useActiveTCP=true) feature=Base
    Waypoint a_frog: TCP in base x=336.638 y=773.336 z=103.937 mm, rx=-1.3698 ry=-2.3362 rz=1.327 rad; joints [-127.102, -6.181, 18.995, -50.118, -88.699, -156.884] deg
      Until EXPRESSION (allowActions=false) ExpressionBranch=beats≥3
  Timer (action=Reset) variable=beats
  MoveL speed 100 mm/s, acceleration 600 mm/s^2 (useActiveTCP=true) feature=Base
    Waypoint a_tip: TCP in base x=525.206 y=350.983 z=214.78 mm, rx=-1.3698 ry=-2.3362 rz=1.327 rad; joints [-161.028, -44.56, 81.191, -78.693, -115.03, -178.818] deg
      Until EXPRESSION (allowActions=false) ExpressionBranch=beats≥3
    Timer (action=Reset) variable=beats
  MoveL speed 100 mm/s, acceleration 600 mm/s^2 (useActiveTCP=true) feature=Base
    Waypoint a_frog: TCP in base x=336.638 y=773.336 z=103.937 mm, rx=-1.3698 ry=-2.3362 rz=1.327 rad; joints [-127.102, -6.181, 18.995, -50.118, -88.699, -156.884] deg
      Until EXPRESSION (allowActions=false) ExpressionBranch=beats≥3
  Timer (action=Reset) variable=beats
  MoveL speed 100 mm/s, acceleration 600 mm/s^2 (useActiveTCP=true) feature=Base
    Waypoint a_tip: TCP in base x=525.206 y=350.983 z=214.78 mm, rx=-1.3698 ry=-2.3362 rz=1.327 rad; joints [-161.028, -44.56, 81.191, -78.693, -115.03, -178.818] deg
      Until EXPRESSION (allowActions=false) ExpressionBranch=beats≥3
    Timer (action=Reset) variable=beats
  MoveL speed 150 mm/s, acceleration 600 mm/s^2 (useActiveTCP=true) feature=Base
    Waypoint a_frog: TCP in base x=336.638 y=773.336 z=103.937 mm, rx=-1.3698 ry=-2.3362 rz=1.327 rad; joints [-127.102, -6.181, 18.995, -50.118, -88.699, -156.884] deg
      Until EXPRESSION (allowActions=false) ExpressionBranch=beats≥3
  Timer (action=Reset) variable=beats
  MoveL speed 100 mm/s, acceleration 600 mm/s^2 (useActiveTCP=true) feature=Base
    Waypoint a_tip: TCP in base x=525.206 y=350.983 z=214.78 mm, rx=-1.3698 ry=-2.3362 rz=1.327 rad; joints [-161.028, -44.56, 81.191, -78.693, -115.03, -178.818] deg
      Until EXPRESSION (allowActions=false) ExpressionBranch=beats≥9.5
    Timer (action=Reset) variable=beats
